{attribute 'GeneratedUsingTerminal: KL3201'}
{attribute addProperty BoxType "KL3201"}
{attribute addProperty Id "Channel_1AT %Q*Channel_6576A6810"}
{attribute addProperty CRC "1632160004"}
{attribute addProperty Size "0"}
TYPE KL3201_6148C904 :
STRUCT
	{attribute addProperty Name "Channel_1"}
	Channel_1 : Channel_6576A681;
END_STRUCT
END_TYPE

(* stored: Version 1.2.0.0, ProductVersion 3.1.4024.9
   DUT KL3201_6148C904: Id {1bf68045-accb-43e7-9c46-ee708853ef09} *)
